{attribute 'qualified_only'}
VAR_GLOBAL
	Inicio:BOOL;
	PesoMaxConte:REAL;
	Dosis:REAL;
	Tinyeccion:DINT;
	PesoBatch:REAL;
	Tolerancia:REAL;
	Pausa:BOOL;		
	Error:REAL;
	ContLleno:BOOL;	
	CantPesadas:INT;
	PesoCalibracion:REAL;
	Muestra1_Ok:BOOL;
	Finalizado:BOOL;
	PesoPromedio6:REAL;
	
END_VAR

(* stored: Version 1.1.0.1, ProductVersion 3.1.4024.14
   GVL HMIcalP1: Id {b2f2f4d0-d15d-4129-a9f7-1ea9d3496a5d} *)
